{attribute 'linkalways'} 
{attribute 'no_explicit_call' := 'This FB is a CLASS and must be accessed using methods or properties'}
{attribute 'enable_dynamic_creation'}
FUNCTION_BLOCK INTERNAL ABSTRACT Mc2MotionCommand EXTENDS Mc2Command IMPLEMENTS MotionCommand
VAR
END_VAR

{attribute 'monitoring' := 'call'}
PROPERTY PUBLIC ABSTRACT Active : BOOL
GET // PUBLIC
END_GET
END_PROPERTY

END_FUNCTION_BLOCK

(* stored: Version 1.1.0.1
   POU Mc2MotionCommand: Id {b9feb950-837c-0c63-3efe-0cf9473a606f}, SpecialFunc None
   Property Active: Id {6e440f34-2bfa-01bb-08ff-9edd6af43fbb}
   Get Get: Id {f0c67215-0008-0488-0c4d-4470e62a6019} *)
